Fanuc KAREL source: V_CAM_CALIB.kl

PROGRAM T
%NOLOCKGROUP
VAR
 v0 : STRING[40]
 v1 : INTEGER
 v2 : INTEGER
BEGIN
 V_CAM_CALIB(v0, v1, v2)
END T
